FUNCTION_BLOCK CarLightCtl_AT (* Function block for controling the operation of a car trafic light following the rules of Germany *)
  (* Standard: 61499-2 *)
  (* Version 0.0, 2014-07-11, 4DIAC-IDE, 4DIAC-Consortium *)
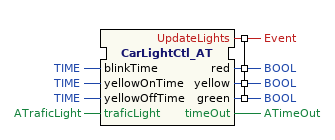
  EVENT_OUTPUT
    UpdateLights WITH green, red, yellow;
  END_EVENT
  VAR_INPUT
    blinkTime : TIME; (* Cycle time for a light blinking(i.e., out of service or switching from green to red) *)
    yellowOnTime : TIME; (* Time the yellow light is on when switching from red to green *)
    yellowOffTime : TIME; (* Time the yellow light is on when swithcing from green to red *)
  END_VAR
  VAR_OUTPUT
    red : BOOL;
    yellow : BOOL;
    green : BOOL;
  END_VAR
  SOCKETS
    traficLight : ATraficLight;
  END_SOCKETS
  PLUGS
    timeOut : ATimeOut;
  END_PLUGS
  VAR
    blinkCount : UINT; (* Internal Variable *)
  END_VAR
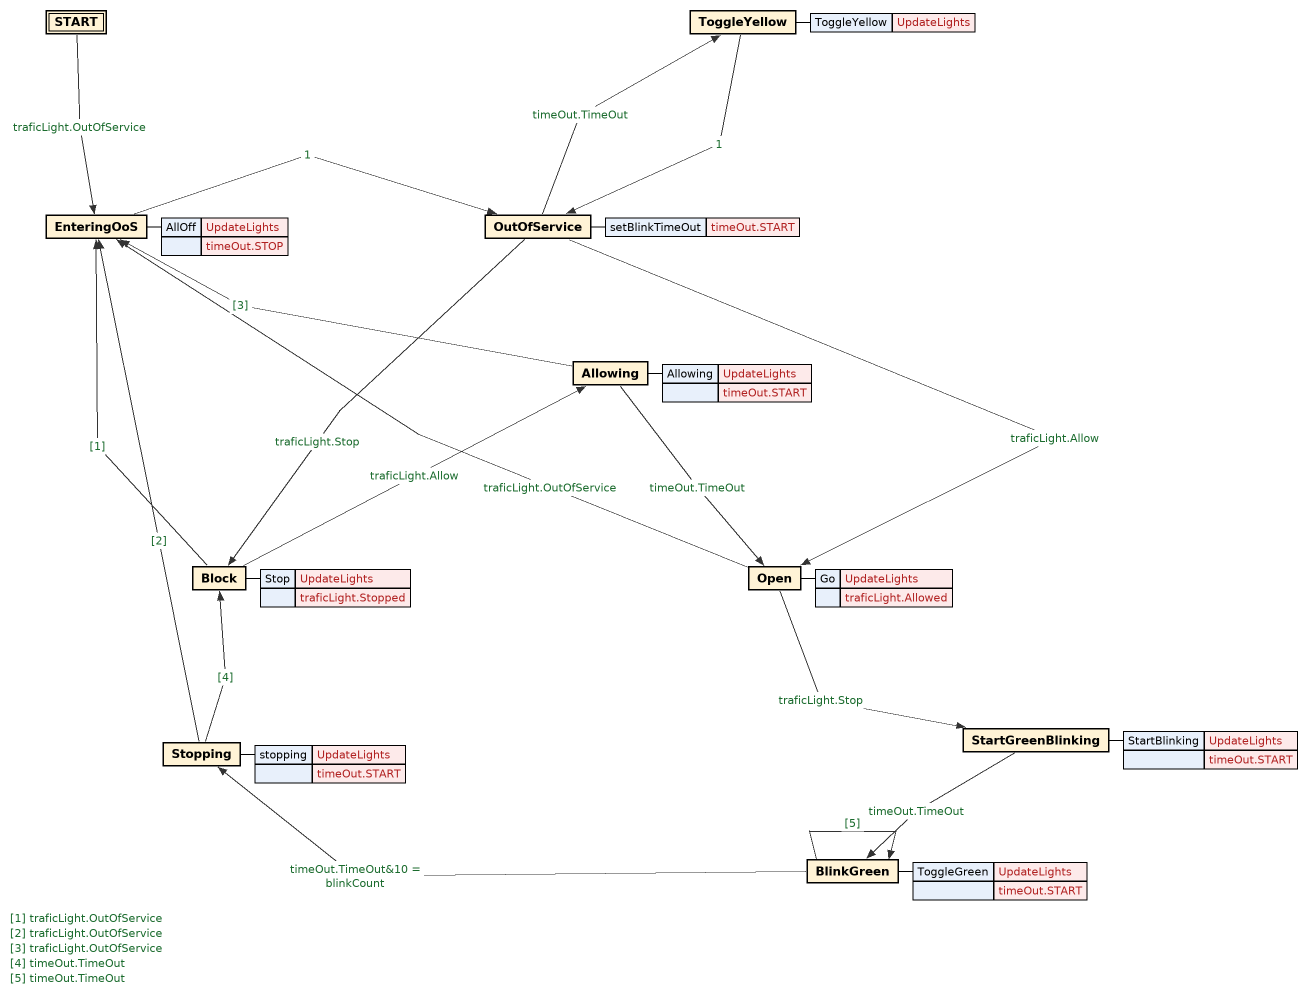
  EC_STATES
    START;
    OutOfService : setBlinkTimeOut -> timeOut.START;
    Block : Stop -> UpdateLights, -> traficLight.Stopped;
    Open : Go -> UpdateLights, -> traficLight.Allowed;
    ToggleYellow : ToggleYellow -> UpdateLights;
    EnteringOoS : AllOff -> UpdateLights, -> timeOut.STOP;
    Allowing : Allowing -> UpdateLights, -> timeOut.START;
    Stopping : stopping -> UpdateLights, -> timeOut.START;
    StartGreenBlinking : StartBlinking -> UpdateLights, -> timeOut.START;
    BlinkGreen : ToggleGreen -> UpdateLights, -> timeOut.START;
  END_STATES
  EC_TRANSITIONS
    OutOfService TO Block := traficLight.Stop;
    OutOfService TO ToggleYellow := timeOut.TimeOut;
    ToggleYellow TO OutOfService := 1;
    START TO EnteringOoS := traficLight.OutOfService;
    Block TO EnteringOoS := traficLight.OutOfService;
    Open TO EnteringOoS := traficLight.OutOfService;
    EnteringOoS TO OutOfService := 1;
    Block TO Allowing := traficLight.Allow;
    Allowing TO Open := timeOut.TimeOut;
    Stopping TO EnteringOoS := traficLight.OutOfService;
    Stopping TO Block := timeOut.TimeOut;
    Allowing TO EnteringOoS := traficLight.OutOfService;
    OutOfService TO Open := traficLight.Allow;
    Open TO StartGreenBlinking := traficLight.Stop;
    StartGreenBlinking TO BlinkGreen := timeOut.TimeOut;
    BlinkGreen TO Stopping := timeOut.TimeOut&10 = blinkCount;
    BlinkGreen TO BlinkGreen := timeOut.TimeOut;
  END_TRANSITIONS
  ALGORITHM AllOff IN ST:
red := FALSE;
yellow := FALSE;
green := FALSE;
  END_ALGORITHM
  ALGORITHM Stop IN ST: (* Put lights in stop mode (i.e., red := true, green := false) *)
red := TRUE;
yellow := FALSE;
green := FALSE;
  END_ALGORITHM
  ALGORITHM Go IN ST: (* Put lights in Walk mode (i.e., red := false, green := true) *)
red := FALSE;
yellow := FALSE;
green := TRUE;
  END_ALGORITHM
  ALGORITHM setBlinkTimeOut IN ST:
timeOut.DT := blinkTime;
  END_ALGORITHM
  ALGORITHM ToggleYellow IN ST: (* new algorithm *)
yellow := NOT yellow;
  END_ALGORITHM
  ALGORITHM Allowing IN ST: (* new algorithm *)
yellow := TRUE;
timeOut.DT := yellowOnTime;
  END_ALGORITHM
  ALGORITHM stopping IN ST: (* new algorithm *)
green := FALSE;
yellow := TRUE;

timeOut.DT := yellowOffTime;
  END_ALGORITHM
  ALGORITHM StartBlinking IN ST: (* new algorithm *)
timeOut.DT := blinkTime;
blinkCount := 0;
green := FALSE;
  END_ALGORITHM
  ALGORITHM ToggleGreen IN ST: (* new algorithm *)
green := NOT green;
blinkCount := blinkCount + 1;
  END_ALGORITHM
END_FUNCTION_BLOCK
